FUNCTION_BLOCK BfbSetterResetter
  (* Standard: 61499-2 *)
  (* Version 0.1, 2019-00-29, hpea485, UOA *)
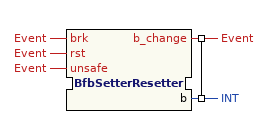
  EVENT_INPUT
    brk;
    rst;
    unsafe;
  END_EVENT
  EVENT_OUTPUT
    b_change WITH b;
  END_EVENT
  VAR_OUTPUT
    b : INT;
  END_VAR
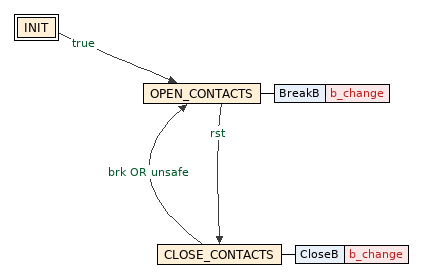
  EC_STATES
    INIT;
    OPEN_CONTACTS : BreakB -> b_change;
    CLOSE_CONTACTS : CloseB -> b_change;
  END_STATES
  EC_TRANSITIONS
    INIT TO OPEN_CONTACTS := true;
    OPEN_CONTACTS TO CLOSE_CONTACTS := rst;
    CLOSE_CONTACTS TO OPEN_CONTACTS := brk OR unsafe;
  END_TRANSITIONS
  ALGORITHM BreakB IN C:
me->b = 1;
  END_ALGORITHM
  ALGORITHM CloseB IN C:
me->b = 0;
  END_ALGORITHM
END_FUNCTION_BLOCK
